// Mitsubishi GX Works2 project: 02102023 CLP aula   PLC: Q03UDV

// global labels: Global1
VAR_GLOBAL
  gi_xSensorTempDoFornoDaSecadora AT X0 : BOOL;  (* Imput 0 do cartão de entrada *)
  g_cValorDaConstante AT YI : ;
  G_xAtuador : ;
END_VAR

// task Task_01 (event TRUE, interval 0, priority 31): POU_01

PROGRAM POU_01
VAR
  CTD_1 : CTD;
  CTUD_1 : CTUD;
  CTUD_2 : CTUD;
  CTUD_E_1 : CTUD_E;
  Contador de processo : ;
  Contadordeprocesso : CTUD;
  Contadordeprocessoqd : INT;
  TP_1 : TP;
  TON_1 : TOF;
  TOF_1 : TOF;
  TimeTP : ;
  TimeON : TIME;
  TimeOFF : TIME;
  TimeTimeTP : TIME;
END_VAR
(* structured ladder/FBD written out as ST: instructions are called as NAME(EN, inputs, outputs); _pN, _eN, _tN stand for wires *)
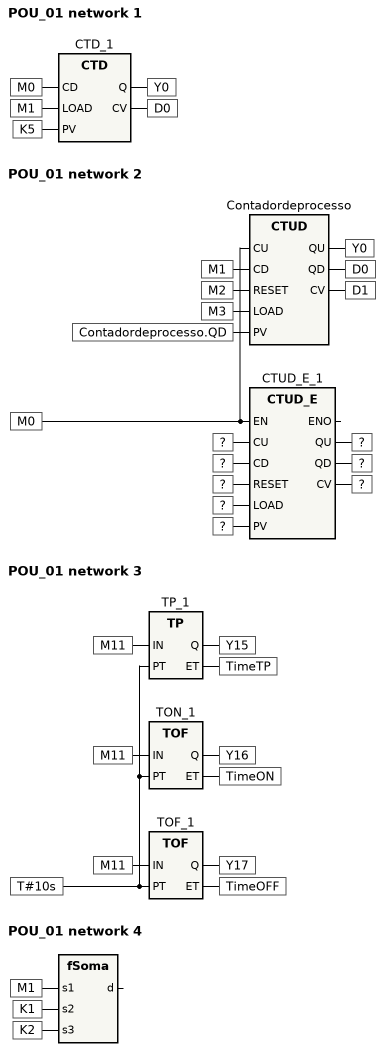
(* network 1 *)
CTD_1(CD := M0, LOAD := M1, PV := K5, Q => Y0, CV => D0);
(* network 2 *)
Contadordeprocesso(CU := M0, CD := M1, RESET := M2, LOAD := M3, PV := Contadordeprocesso.QD, QU => Y0, QD => D0, CV => D1);
CTUD_E_1(EN := M0, CU := ?, CD := ?, RESET := ?, LOAD := ?, PV := ?, QU => ?, QD => ?, CV => ?);
(* network 3 *)
TP_1(IN := M11, PT := T#10s, Q => Y15, ET => TimeTP);
TON_1(IN := M11, PT := T#10s, Q => Y16, ET => TimeON);
TOF_1(IN := M11, PT := T#10s, Q => Y17, ET => TimeOFF);
(* network 4 *)
fSoma(M1, K1, K2);
END_PROGRAM

FUNCTION fSoma
VAR_INPUT
  i_xHabilitar : ;
  i_iElemento1 : INT;
  i_iElemento2 : INT;
END_VAR
(* structured ladder/FBD written out as ST: instructions are called as NAME(EN, inputs, outputs); _pN, _eN, _tN stand for wires *)
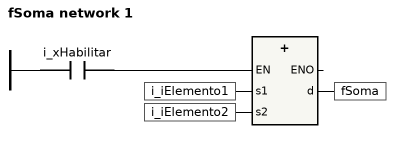
(* network 1 *)
+(i_xHabilitar, i_iElemento1, i_iElemento2, fSoma);
END_FUNCTION

FUNCTION fSubtracaoInt
VAR_INPUT
  i_xEnable : INT;
  i_xElement1 : INT;
  i_xElement2 : INT;
END_VAR
(* structured ladder/FBD written out as ST: instructions are called as NAME(EN, inputs, outputs); _pN, _eN, _tN stand for wires *)
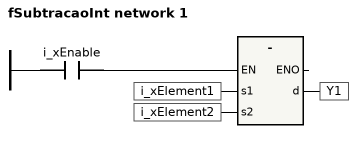
(* network 1 *)
-(i_xEnable, i_xElement1, i_xElement2, Y1);
END_FUNCTION

FUNCTION iProdutoInt
VAR_INPUT
  i_xProduto : INT;
  i_xElemento2 : INT;
  i_xElemento1 : INT;
END_VAR
(* structured ladder/FBD written out as ST: instructions are called as NAME(EN, inputs, outputs); _pN, _eN, _tN stand for wires *)
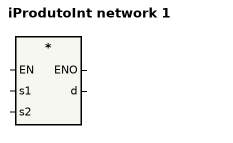
(* network 1 *)
*(_open, _open, _open, _open);
END_FUNCTION

FUNCTION fQuociente
VAR_INPUT
  i_xDividir : INT;
  i_iDivisor : INT;
  i_iDividendo : INT;
END_VAR
(* structured ladder/FBD written out as ST: instructions are called as NAME(EN, inputs, outputs); _pN, _eN, _tN stand for wires *)
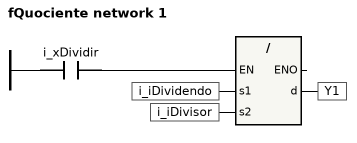
(* network 1 *)
/(i_xDividir, i_iDividendo, i_iDivisor, Y1);
END_FUNCTION

FUNCTION_BLOCK fbBlinker
VAR_INPUT
  i_xEnable : BOOL;
  i_tHightPulse : TIME;
  i_tLowPulse : TIME;
END_VAR
VAR_OUTPUT
  o_xPulse : BOOL;
END_VAR
VAR
  fb TimerHigh : TP;
  fb TimerLow : TOF;
  xAuxilar : BOOL;
  fbTimerHigh : TP;
END_VAR
(* structured ladder/FBD written out as ST: instructions are called as NAME(EN, inputs, outputs); _pN, _eN, _tN stand for wires *)
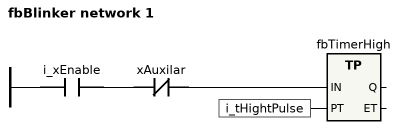
(* network 1 *)
fbTimerHigh(IN := i_xEnable AND NOT xAuxilar, PT := i_tHightPulse);
END_FUNCTION_BLOCK
